
FUNCTION CB_bool_to_dword : DWORD

TITLE = ' Convert a boolean into an double word '
VERSION : '1.0'
AUTHOR  : CB
NAME    : boToDwor
FAMILY  : TNI

VAR_INPUT
    IN : BOOL;
END_VAR

VAR_TEMP

END_VAR

BEGIN

CB_bool_to_dword := DINT_TO_DWORD(BOOL_TO_DINT(IN));

END_FUNCTION
